// This function has been automatically generated from the project information.
{attribute 'signature_flag' := '1073741824'}
{attribute 'TcGenerated'}
{attribute 'no-analysis'}
FUNCTION F_GetCompany : WSTRING
VAR_INPUT
	
END_VAR

F_GetCompany := "RKe";

END_FUNCTION

(* stored: Version 1.1.0.1
   POU F_GetCompany: Id {abe5afb3-0c2b-444a-ac06-bb982f3e01ec}, SpecialFunc None *)
